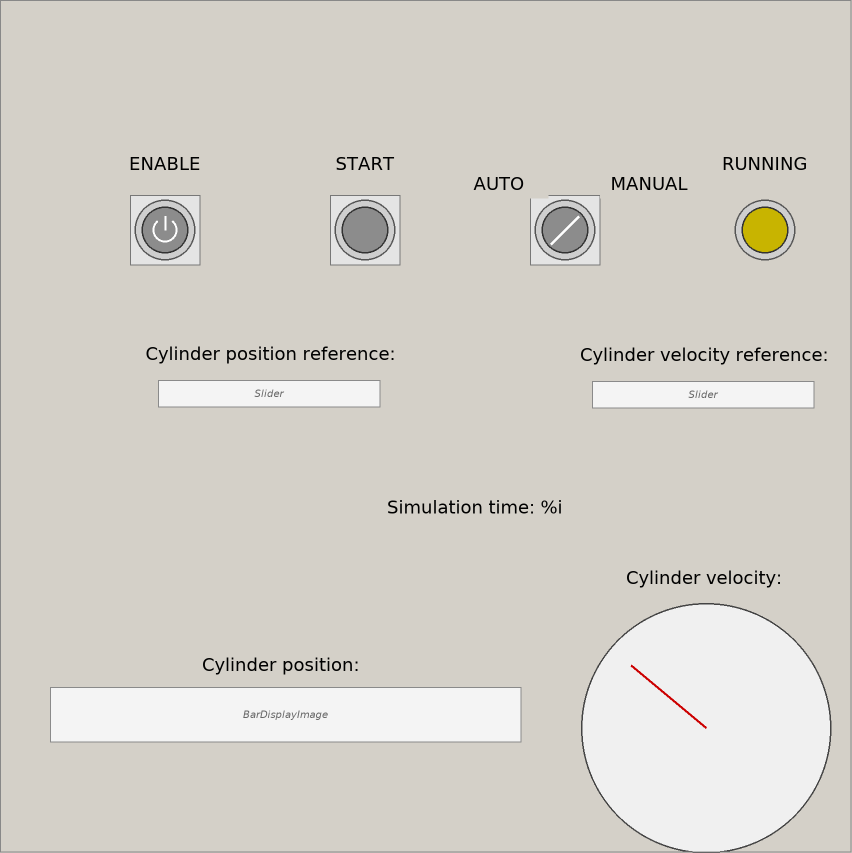
VISUALIZATION CraneHMI  // 852x853
    PowerSwitch (130,195 70x70), variable: Inputs.bEnableSimulation, behaviour: TOGGLE, style: Switch-PowerSwitch-Gray
    RotarySwitch (530,195 70x70), variable: Inputs.bAutoMode, behaviour: TOGGLE, style: Switch-RotarySwitch-Gray
    PushSwitch (330,195 70x70), variable: Inputs.bStartSimulation, behaviour: TOGGLE, style: Switch-PushSwitch-Gray
    Rectangle (115,150 100x28), "ENABLE"
    Rectangle (315,150 100x28), "START"
    Rectangle (450,170 98x28), "AUTO"
    Rectangle (600,170 98x28), "MANUAL"
    Lamp1 (730,195 70x70), variable: Inputs.bEnableSimulation, style: Lamp-Lamp1-Yellow
    Rectangle (715,150 100x28), "RUNNING"
    BarDisplayImage (50,687 471x55), value: Outputs.fCylinderPosition, style: BarDisplayImage-Gray, scale format: %.1f, scale 0..20
    Rectangle (207,494 536x27), "Simulation time: %i", text variable: Outputs.fSimulationTime
    Meter360 (581,603 250x250), value: Outputs.fCylinderVelocity, style: Meter-Meter360-Gray, scale format: %.1f, scale -3..3
    Rectangle (192,652 178x26), "Cylinder position:"
    Rectangle (615,565 178x26), "Cylinder velocity:"
    Slider (158,380 222x27), variable: Inputs.fManualCylinderPositionReference, scale 0..20
    Rectangle (123,342 295x24), "Cylinder position reference:"
    Slider (592,381 222x27), variable: Inputs.fCylinderVelocityReference, scale -3..3
    Rectangle (557,343 295x24), "Cylinder velocity reference:"
END_VISUALIZATION

(* stored: Version 1.1.0.1, ProductVersion 3.1.4024.10
   Visu CraneHMI: Id {b5520909-ac3e-4cb2-bbd3-14e4794d6a77} *)
